{attribute 'qualified_only'}
{attribute 'strict'}
TYPE ChannelType :
(
	NONE := Tc2_PlcInterpolation.E_ItpChannelType.ItpChannelTypeNone,
	INTERPRETER := Tc2_PlcInterpolation.E_ItpChannelType.ItpChannelTypeInterpreter,
	KINEMATIC := Tc2_PlcInterpolation.E_ItpChannelType.ItpChannelTypeKinematic,
	INVALID_ITF_VERSION := Tc2_PlcInterpolation.E_ItpChannelType.ItpChannelType_InvalidItfVer
) INT;
END_TYPE

(* stored: Version 1.1.0.1, ProductVersion 3.1.4024.12
   DUT ChannelType: Id {e8df33f8-a9ee-032c-2457-afa9ef326e25} *)
